ABB RobotStudio station: practica3.rsstn

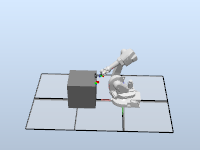
Station practica3 (saved by RobotStudio 20.4.9280.0)
Controller Controlador4
  mechanical unit ROB_1: IRB1600_6_145__02, 6 joints, base frame (0, 0, 0) mm
Layout (positions relative to the parent item):
  - IRB1600_6_145__02 [mechanism, from Robots\IRB1600_6_145_G_02.rslib] at (0, 0, 0) mm; joint values [0.326, -0.2862, 0.8219, -0.4788, 0.4423, 0.699] (rad or m)
  - MyTool [mechanism, from Training Objects\myTool.rslib] at (483.67, 150, 800.53) mm, rotated rx -180 ry 38 rz -180 deg
  - Pieza_1 [part]
Attachment: MyTool is attached to IRB1600_6_145__02 / Link6
Targets, tools, work objects and paths stored in the station, written as RAPID:
! task T_ROB1
MODULE CalibData
  PERS tooldata MyTool:=[TRUE,[[31.792631019,0,229.638935148],[0.945518576,0,0.325568154,0]],[1,[0,0,1],[1,0,0,0],0,0,0]];
ENDMODULE

! task T_ROB1
MODULE Module1
  CONST robtarget pInicio:=[[600,150,600],[0,0,1,0],[0,0,0,0],[9E+09,9E+09,9E+09,9E+09,9E+09,9E+09]];
  PROC Path_10()
    MoveL pInicio,v1000,z100,MyTool\WObj:=wobj0;
  ENDPROC
ENDMODULE

